FUNCTION CheckCritical : BOOL
VAR_INPUT
END_VAR
VAR
END_VAR

CheckCritical := 
    NOT GVL_FSM.sdc_closed OR
    GVL_PT.ERROR_STATUS <> 0 OR
    GVL_PT.MAX_TEMP > GVL_FSM.critical_temp OR
    GVL_Levi.levitation_fault OR
    GVL_Prop.propulsion_fault;

END_FUNCTION

(* stored: Version 1.1.0.1
   POU CheckCritical: Id {b7f02efc-5073-4782-bdb4-49dadea447fc}, SpecialFunc None *)
